# EPICS substitutions: ghosts_data.subs
file pacman_game_parameter.template
{ pattern
  { NAME,	DEVICE,	P,	DRVH,	DRVL,	VAL	}
}
